FUNCTION F_OpenDialog : BOOL
VAR_INPUT
	sDialogName : STRING;
END_VAR
VAR
	pstClientData : POINTER TO VisuElems.VisuStructClientData;
	itfDialogManager : VisuElems.IDialogManager;
	itfMyDialog : VisuElems.IVisualisationDialog;
	stVisuRect : VisuElems.VisuStructSimpleRectangle;
END_VAR

VisuElems.VisuElemBase.g_ClientManager.BeginIteration();
pstClientData := VisuElems.VisuElemBase.g_ClientManager.GetNextClient();
WHILE pstClientData <> 0 DO
   IF pstClientData^.GlobalData.ClientType = VisuElems.Visu_ClientType.HMITargetVisualization THEN
      itfDialogManager := VisuElems.g_VisuManager.GetDialogManager();
      itfMyDialog := itfDialogManager.GetDialog(sDialogName);
      stVisuRect.ptTopLeft.iX := ANY_TO_INT(INT#0);
      stVisuRect.ptTopLeft.iY := ANY_TO_INT(INT#0);
      stVisuRect.ptBottomRight.iX := ANY_TO_INT(10);
      stVisuRect.ptBottomRight.iY := ANY_TO_INT(10);
      itfDialogManager.OpenDialog(itfMyDialog, pstClientData, FALSE, ADR(stVisuRect));
   END_IF
   pstClientData := VisuElems.VisuElemBase.g_ClientManager.GetNextClient();
END_WHILE

END_FUNCTION

(* stored: Version 1.1.0.1, ProductVersion 3.1.4024.9
   POU F_OpenDialog: Id {3b8de8e6-0577-4bd5-86fd-7a5e7f633374}, SpecialFunc None *)
